FUNCTION_BLOCK Q_NumericValueAux (* Command change numeric value ( Part 6 - F.22 ) *)
  (* Standard: ISO 11783-6; Description: Copyright (c) 2022 HR Agrartechnik GmbH This program and the accompanying materials are made available under the terms of the Eclipse Public License 2.0 which is available at https://www.eclipse.org/legal/epl-2.0/ SPDX-License-Identifier: EPL-2.0 see Description Tab *)
  (* Version 1.0, 2022-07-08, Franz Höpfinger, HR Agrartechnik GmbH *)
  (* Documentation:
  Command change numeric value ( Part 6 - F.22 )
   This command is used to change the value of an object. It applies only to objects that have a numeric value attribute.
   param[in] {objectID, uint16_t}
   Object ID
   param[in] {value, uint32_t}
   New value of ID
   Return Values: 
   int16_t
    - VT_E_NO_ERR (0) - OK
   - VT_E_OVERFLOW (-6) - buffer overflow
   - VT_E_NOACT (-8) - Command not possible in current state
   - VT_E_NO_INSTANCE (-21) - No VT client available
   - VT_E_ISO_INSTANCE_INVALID (-129) - Identifier for instance (connection) invalid
   - VT_E_HANDLE_INVALID (-128) - ErrorCause: invalid Handle
   - VT_E_NOT_ALIVE (-130) - Identifier for instance valid, but VT Dead.
  *)
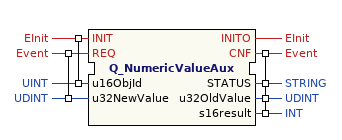
  EVENT_INPUT
    INIT : EInit WITH u16ObjId; (* Service Initialization *)
    REQ WITH u32NewValue; (* Service Request *)
  END_EVENT
  EVENT_OUTPUT
    INITO : EInit; (* Initialization Confirm *)
    CNF WITH STATUS, u32OldValue, s16result; (* Confirmation of Requested Service *)
  END_EVENT
  VAR_INPUT
    u16ObjId : UINT; (* Object ID *)
    u32NewValue : UDINT; (* New value of ID *)
  END_VAR
  VAR_OUTPUT
    STATUS : STRING; (* Service Status *)
    u32OldValue : UDINT; (* Old value of ID *)
    s16result : INT; (* retval see description *)
  END_VAR
END_FUNCTION_BLOCK
